(* CODESYS project ludo.ecp

Project tree, tasks and I/O mapping:
  Controller : 750-8214 PFC200 G2 2ETH RS CAN, WAGO, order no. 0750-8214, version 5.15.4.20
    application Application
      libraries: 
      task PLC_Task (cyclic, interval t#50ms, priority 15) calls PLC_PRG
      program POU [SFC]: Step0_active
      function block can_hit_opponent [ST]
      function all_token_home [ST]
      function any_token_home [ST]
    Kbus : Kbus, WAGO, version 1.4.0.2
        unmapped channels: K-BUS diagnostics
    MODBUS
      MODBUS : MODBUS, WAGO, order no. n/a, version 1.1.1.15
    CANbus
    Common.PCI
    Serial
      COM1 : COM1, WAGO, version 0.0.0.19
*)

// Controller/Application/POU
PROGRAM POU
VAR
	dice_val: UINT;
	can_hit_opponent_0: can_hit_opponent;
	position: UINT;
	robot_positions: ARRAY [0..3] OF INT;
	human_positions: ARRAY [0..11] OF INT;
	button_pressed: BOOL;
	can_hit_opponent0: can_hit_opponent;
	can_hit_opponent_bool: BOOL;
END_VAR

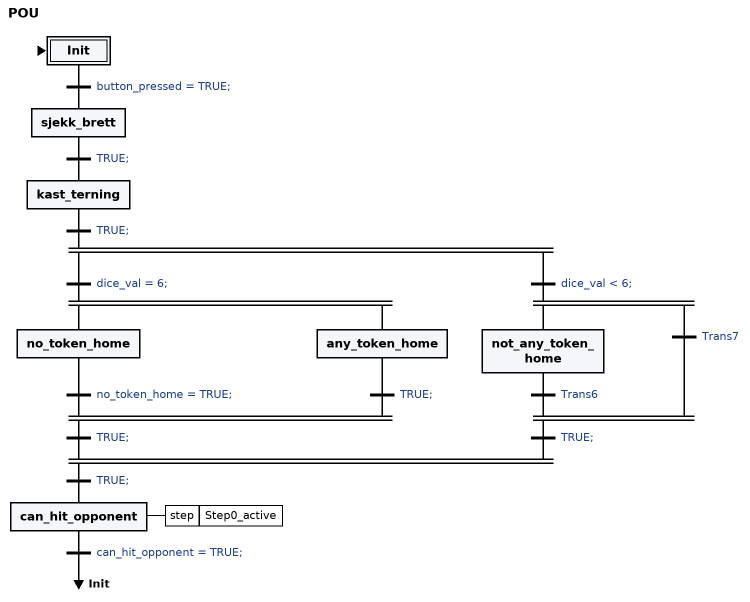
INITIAL_STEP Init:
END_STEP
TRANSITION FROM Init TO sjekk_brett
    := button_pressed = TRUE;
END_TRANSITION
STEP sjekk_brett:
END_STEP
TRANSITION FROM sjekk_brett TO kast_terning
    := TRUE;
END_TRANSITION
STEP kast_terning:
END_STEP
TRANSITION FROM kast_terning TO (???, ???)
    := TRUE;
END_TRANSITION
TRANSITION FROM ??? TO (no_token_home, any_token_home)
    := dice_val = 6;
END_TRANSITION
STEP no_token_home:
END_STEP
TRANSITION FROM no_token_home TO ???
    := no_token_home = TRUE;
END_TRANSITION
STEP any_token_home:
END_STEP
TRANSITION FROM any_token_home TO ???
    := TRUE;
END_TRANSITION
TRANSITION FROM (???, ???) TO ???
    := TRUE;
END_TRANSITION
TRANSITION FROM ??? TO (not_any_token_home, ???)
    := dice_val < 6;
END_TRANSITION
STEP not_any_token_home:
END_STEP
TRANSITION FROM not_any_token_home TO ???
    := Trans6;
END_TRANSITION
TRANSITION FROM ??? TO ???
    := Trans7;
END_TRANSITION
TRANSITION FROM (???, ???) TO ???
    := TRUE;
END_TRANSITION
TRANSITION FROM (???, ???) TO can_hit_opponent
    := TRUE;
END_TRANSITION
STEP can_hit_opponent:
    Step0_active(N);  // step action
END_STEP
TRANSITION FROM can_hit_opponent TO Init
    := can_hit_opponent = TRUE;
END_TRANSITION

ACTION Step0_active:
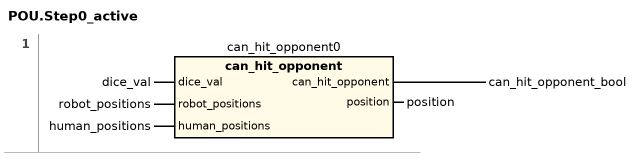
// NETWORK 1
can_hit_opponent0(
    dice_val := dice_val,
    robot_positions := robot_positions,
    human_positions := human_positions,
    position => position); // can_hit_opponent
can_hit_opponent_bool := can_hit_opponent0.can_hit_opponent;
END_ACTION

END_PROGRAM

// Controller/Application/can_hit_opponent
FUNCTION_BLOCK can_hit_opponent
VAR_INPUT
	dice_val: UINT;
	robot_positions: ARRAY[0..3] OF INT;
	human_positions: ARRAY[0..11] OF INT;
END_VAR
VAR_OUTPUT
	can_hit_opponent: BOOL;
	position: UINT;
END_VAR
VAR
	human_position: UINT;
	robot_position: UINT;
	i: UINT;
	n: UINT;
END_VAR

FOR i:= 0 TO SIZEOF(robot_positions) - 1 BY 1 DO
	FOR n := 0 TO SIZEOF(human_positions) - 1 BY 1 DO
		IF robot_position[i] + dice_val = human_position[n] THEN
			position:= robot_position[i];
			RETURN;
		END_IF
	END_FOR
END_FOR

END_FUNCTION_BLOCK

// Controller/Application/all_token_home
FUNCTION all_token_home : BOOL
VAR_INPUT
	robot_positions: ARRAY[0..3] OF INT;
END_VAR
VAR
	i: UINT;
END_VAR

FOR i:= 0 TO SIZEOF(robot_positions) - 1 BY 1 DO
	IF robot_positions[i] > 3 THEN
		all_token_home := FALSE;
		RETURN;
	END_IF
END_FOR

END_FUNCTION

// Controller/Application/any_token_home
FUNCTION any_token_home : BOOL
VAR_INPUT
	robot_positions: ARRAY[0..3] OF INT;
END_VAR
VAR
	i: UINT;
END_VAR

FOR i:= 0 TO SIZEOF(robot_positions) - 1 BY 1 DO
	IF robot_positions[i] <= 3 THEN
		any_token_home := TRUE;
		RETURN;
	END_IF
END_FOR

END_FUNCTION
